ABB RobotStudio station: RS2_Picker.rsstn

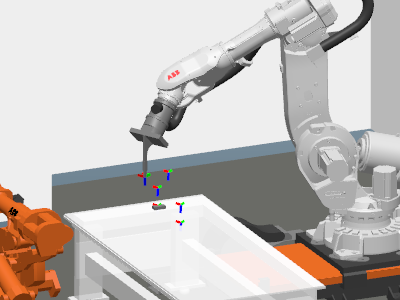
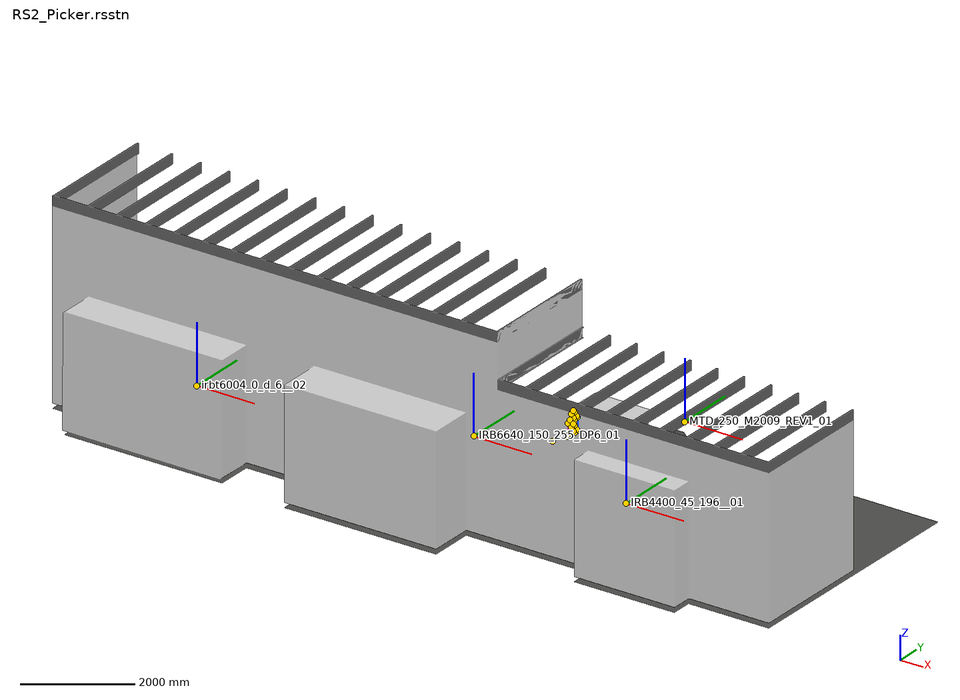
[picture v1: parts stored in the station drawn from their meshes, with robot base, taught points and paths (robot models come from the ABB library and are not in the file)]
Station RS2_Picker (saved by RobotStudio 22.2.9947.0)
Controller dFAB4400, task T_ROB1: task frame (RAPID world) sits at (8239.64, -6.06, -391.24) mm, rotated rx 0 ry 0 rz 180 deg in the station
Controller 66-101898AOFFLINE
  mechanical unit TRACK_1: irbt6004_0_d_6__02, 1 joints, base frame (0, 0, 0) mm
  mechanical unit ROB_1: IRB6640_150_255_DP6_01, 6 joints, base frame (0, 0, 0) mm
Controller dFAB4400
  mechanical unit STN1: MTD_250_M2009_REV1_01, 1 joints, base frame (1410.71, 486.5, 778.9) mm, rotated rx 0 ry 0 rz 90 deg
  mechanical unit ROB_1: IRB4400_45_196__01, 6 joints, base frame (0, 0, 0) mm
Layout (positions relative to the parent item):
  - irbt6004_0_d_6__02 [mechanism, from Libraries\irbt6004_0_d_6__02.rslib] at (-550.5, -475, -384.5) mm; joint values [5] (rad or m)
  - IRB6640_150_255_DP6_01 [mechanism, from Libraries\IRB6640_150_255_DP6_G_01.rslib] at (5000, 0, 0) mm; joint values [-0.2102, 0.1488, 0.3671, 0.9174, 0.6091, -0.3077] (rad or m)
  - rotary_stand [part], size 301.9 x 311.7 x 727.3 mm
  - MTD_250_M2009_REV1_01 [mechanism, from Libraries\MTD_250_M2009_REV1_01.rslib] at (8228.8, 1787.55, 468) mm, rotated rx 0 ry 0 rz 90 deg; joint values [0] (rad or m)
  - IRB4400_45_196__01 [mechanism, from Robots\IRB4400_45_196__01.rslib] at (8239.64, -6.06, -391.24) mm, rotated rx 0 ry 0 rz 180 deg; joint values [1.5707, -1.1345, 0, 0, 0, 0] (rad or m)
  - aarl_floor [part] at (0, 0, -101) mm, size 15367 x 6261.1 x 0 mm
  - 4400 ATI [part] at (8239.59, -419.45, 814.89) mm, rotated rx 0 ry 90 rz -90.01 deg, size 369.5 x 443 x 336 mm
  - AARL_Walls_west [part], size 15367 x 3481.8 x 3810 mm
  - AARL_Walls_east [part], size 15367 x 2779.3 x 3810 mm
  - AARL_Ceiling_west [part], size 15214.6 x 2567.4 x 1117.6 mm
  - VaccumTable_AtEndOfTrack [part], size 1240.6 x 2443.9 x 841 mm
  - ExpanderStation [part], size 715.1 x 918.2 x 79.1 mm
  - Component_SteelTable_2015_10_31 [part] at (1803.71, -1743.4, 287.57) mm, rotated rx 0.58 ry -0.13 rz 179.69 deg, size 2772.7 x 1553.5 x 641.4 mm
  - 20151025_RobotBar_2 [part] at (10163.42, -1202.89, 872.63) mm, rotated rx -90.3 ry 0.37 rz -90.64 deg, size 3760 x 1271.6 x 704 mm
  - 20151107_6640Table_andAlcove [part] at (1803.71, -1743.4, 287.57) mm, rotated rx 0.58 ry -0.13 rz 179.69 deg, size 3362 x 1558.7 x 2265 mm
  - Cameras In Alcove [part], size 3672.3 x 1646.1 x 329.3 mm
  - 6640 ATI [part] at (6755.25, -212.35, 1206.62) mm, rotated rx 139.11 ry 20.7 rz 140.14 deg, size 185.4 x 185.4 x 86.9 mm
  - suctionGripperTool [mechanism] at (6755.25, -212.35, 1206.62) mm, rotated rx 139.11 ry 20.7 rz 140.14 deg
      TCP suctionGripperTool at (-65.22, 118.54, 382.24) mm, rotated rx -42.17 ry -15.36 rz 13.49 deg
      links: Dummy
  - Part_1 [part] at (6893.07, 6354.78, 0) mm, rotated rx 0 ry 0 rz -90.01 deg, size 50 x 100 x 25 mm
  - ITARF23_Pincher [mechanism] at (6755.25, -212.35, 1206.62) mm, rotated rx -139.11 ry -20.7 rz -39.86 deg
      TCP ITARF23_Pincher at (-65.22, 118.54, 382.24) mm, rotated rx -42.17 ry -15.36 rz 13.49 deg
      links: pincherTool
Attachment: IRB6640_150_255_DP6_01 is attached to irbt6004_0_d_6__02 / Link1
Attachment: 4400 ATI is attached to IRB4400_45_196__01 / Link6
Attachment: 6640 ATI is attached to IRB6640_150_255_DP6_01 / Link6
Attachment: suctionGripperTool is attached to IRB6640_150_255_DP6_01 / Link6
Attachment: ITARF23_Pincher is attached to IRB6640_150_255_DP6_01 / Link6
Collision set CollisionSet_1: 4400 ATI against Link4, Link2, near miss 0 m
Collision set CollisionSet_2: 20151025_RobotBar_2 against IRB4400_45_196__01, near miss 0.005 m
Collision set CollisionSet_3: 20151107_6640Table_andAlcove, Component_SteelTable_2015_10_31, ExpanderStation against IRB6640_150_255_DP6_01, near miss 0.005 m
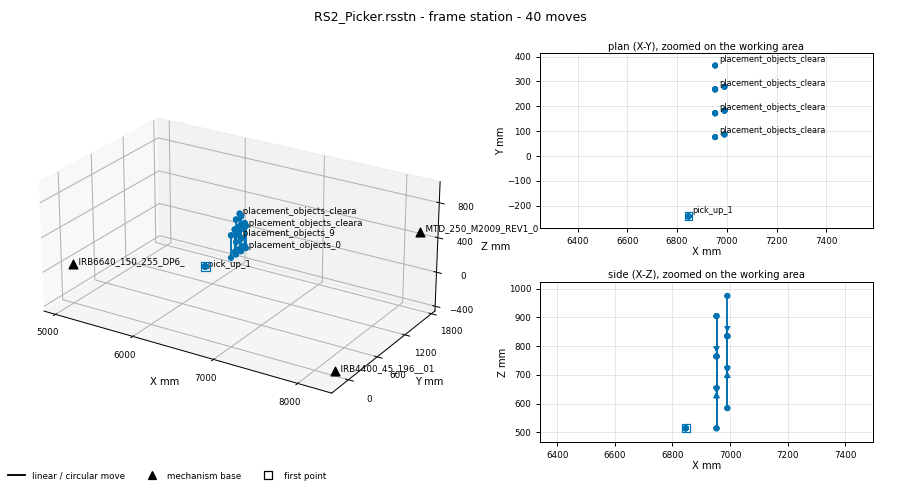
[picture p0: tool path of RS2_Picker.rsstn in frame station, 40 of 72 moves have a stored position in this frame; points joined in program order, loops and branches not executed]
Targets, tools, work objects and paths stored in the station, written as RAPID:
! task T_ROB1
MODULE Inc_Form_Test_090816
  VAR speeddata mySpeed:=[250,250,5000,1000];
  VAR zonedata myZone:=[FALSE,5,5,10,5,10,3];
ENDMODULE

! task T_ROB1
MODULE RobotProgramModule
  CONST robtarget t_pick:=[[6693.807660738,-323.119608005,453.981396454],[0.055399765,0.879680571,-0.471265936,0.031644522],[-1,0,-3,0],[4333.256617002,9E+09,9E+09,9E+09,9E+09,9E+09]];
  CONST robtarget t_pick_safe:=[[6693.807675418,-323.1195903,606.653821091],[0.055399731,0.879680578,-0.471265927,0.031644523],[-1,0,-2,0],[4333.256617002,9E+09,9E+09,9E+09,9E+09,9E+09]];
  CONST robtarget t_place_safe:=[[6693.807761035,133.958968301,606.65379018],[0.05539974,0.879680599,-0.471265883,0.031644591],[0,-1,-2,0],[4333.256617002,9E+09,9E+09,9E+09,9E+09,9E+09]];
  CONST robtarget t_place:=[[6693.80755977,133.959044617,452.547726462],[0.055399551,0.879680524,-0.471266043,0.031644636],[0,-1,-2,0],[4333.256617002,9E+09,9E+09,9E+09,9E+09,9E+09]];
  CONST robtarget t_home:=[[6693.807553504,-112.078129424,808.817014857],[0.055399679,0.879680616,-0.471265852,0.031644705],[-1,0,-2,0],[4333.256617002,9E+09,9E+09,9E+09,9E+09,9E+09]];
ENDMODULE

! task T_ROB1
MODULE CalibData
  PERS tooldata ITARF23_Pincher:=[TRUE,[[-65.2151,118.542,382.236],[0.180955748,0.120020452,-0.358114493,-0.908077155]],[1,[0,0,1],[1,0,0,0],0,0,0]];
ENDMODULE

! task T_ROB1
MODULE MainModule
  PERS tooldata two_finger_gripper_itar2:=[TRUE,[[94.35,-163.419,405.705],[-0.239118,0.099041,-0.369628,0.892406]],[0.001,[0,0,0.001],[1,0,0,0],0,0,0]];
  VAR jointtarget pos_home:=[[1,2,3,4,5,6],[4200,9E+09,9E+09,9E+09,9E+09,9E+09]];
  VAR robtarget pick_up_1:=[[6845.94,-242.64,514.59],[0,0.707107,-0.707107,0],[0,0,0,0],[5000,9E+09,9E+09,9E+09,9E+09,9E+09]];
  VAR robtarget placement_objects_clearance_0:=[[6952.98,364.03,764.59],[0,0.707107,-0.707107,0],[0,0,0,0],[5000,9E+09,9E+09,9E+09,9E+09,9E+09]];
  VAR robtarget placement_objects_0:=[[6952.98,364.03,514.59],[0,0.707107,-0.707107,0],[0,0,0,0],[5000,9E+09,9E+09,9E+09,9E+09,9E+09]];
  VAR robtarget placement_objects_clearance_1:=[[6952.98,268.03,764.59],[0,0.707107,-0.707107,0],[0,0,0,0],[5000,9E+09,9E+09,9E+09,9E+09,9E+09]];
  VAR robtarget placement_objects_1:=[[6952.98,268.03,514.59],[0,0.707107,-0.707107,0],[0,0,0,0],[5000,9E+09,9E+09,9E+09,9E+09,9E+09]];
  VAR robtarget placement_objects_clearance_2:=[[6952.98,172.03,764.59],[0,0.707107,-0.707107,0],[0,0,0,0],[5000,9E+09,9E+09,9E+09,9E+09,9E+09]];
  VAR robtarget placement_objects_2:=[[6952.98,172.03,514.59],[0,0.707107,-0.707107,0],[0,0,0,0],[5000,9E+09,9E+09,9E+09,9E+09,9E+09]];
  VAR robtarget placement_objects_clearance_3:=[[6952.98,76.03,764.59],[0,0.707107,-0.707107,0],[0,0,0,0],[5000,9E+09,9E+09,9E+09,9E+09,9E+09]];
  VAR robtarget placement_objects_3:=[[6952.98,76.03,514.59],[0,0.707107,-0.707107,0],[0,0,0,0],[5000,9E+09,9E+09,9E+09,9E+09,9E+09]];
  VAR robtarget placement_objects_clearance_4:=[[6990.48,278.53,834.59],[0,1,0,0],[0,0,0,0],[5000,9E+09,9E+09,9E+09,9E+09,9E+09]];
  VAR robtarget placement_objects_4:=[[6990.48,278.53,584.59],[0,1,0,0],[0,0,0,0],[5000,9E+09,9E+09,9E+09,9E+09,9E+09]];
  VAR robtarget placement_objects_clearance_5:=[[6990.48,182.53,834.59],[0,1,0,0],[0,0,0,0],[5000,9E+09,9E+09,9E+09,9E+09,9E+09]];
  VAR robtarget placement_objects_5:=[[6990.48,182.53,584.59],[0,1,0,0],[0,0,0,0],[5000,9E+09,9E+09,9E+09,9E+09,9E+09]];
  VAR robtarget placement_objects_clearance_6:=[[6990.48,86.53,834.59],[0,1,0,0],[0,0,0,0],[5000,9E+09,9E+09,9E+09,9E+09,9E+09]];
  VAR robtarget placement_objects_6:=[[6990.48,86.53,584.59],[0,1,0,0],[0,0,0,0],[5000,9E+09,9E+09,9E+09,9E+09,9E+09]];
  VAR robtarget placement_objects_clearance_7:=[[6952.98,268.03,904.59],[0,0.707107,-0.707107,0],[0,0,0,0],[5000,9E+09,9E+09,9E+09,9E+09,9E+09]];
  VAR robtarget placement_objects_7:=[[6952.98,268.03,654.59],[0,0.707107,-0.707107,0],[0,0,0,0],[5000,9E+09,9E+09,9E+09,9E+09,9E+09]];
  VAR robtarget placement_objects_clearance_8:=[[6952.98,172.03,904.59],[0,0.707107,-0.707107,0],[0,0,0,0],[5000,9E+09,9E+09,9E+09,9E+09,9E+09]];
  VAR robtarget placement_objects_8:=[[6952.98,172.03,654.59],[0,0.707107,-0.707107,0],[0,0,0,0],[5000,9E+09,9E+09,9E+09,9E+09,9E+09]];
  VAR robtarget placement_objects_clearance_9:=[[6990.48,182.53,974.59],[0,1,0,0],[0,0,0,0],[5000,9E+09,9E+09,9E+09,9E+09,9E+09]];
  VAR robtarget placement_objects_9:=[[6990.48,182.53,724.59],[0,1,0,0],[0,0,0,0],[5000,9E+09,9E+09,9E+09,9E+09,9E+09]];
  PROC new_pincher()
    ConfJ \On;
    MoveAbsJ pos_home,v200,z50,two_finger_gripper_itar2\WObj:=wobj0;
    ConfJ \Off;
    ConfJ \On;
    MoveAbsJ pos_home,v200,z50,two_finger_gripper_itar2\WObj:=wobj0;
    ConfJ \Off;
    WaitTime 1;
    SetDO do_tool_gripper_close,0;
    SetDO do_tool_gripper_open,1;
    WaitTime 2;
    MoveJ il_21,v300,z15,two_finger_gripper_itar2\WObj:=wobj0;
    MoveL pick_up_1,v300,z0,two_finger_gripper_itar2\WObj:=wobj0;
    WaitTime 1;
    SetDO do_tool_gripper_close,1;
    SetDO do_tool_gripper_open,0;
    WaitTime 2;
    MoveJ il_22,v300,z15,two_finger_gripper_itar2\WObj:=wobj0;
    MoveL placement_objects_clearance_0,v300,z0,two_finger_gripper_itar2\WObj:=wobj0;
    MoveL placement_objects_0,v300,z0,two_finger_gripper_itar2\WObj:=wobj0;
    WaitTime 1;
    SetDO do_tool_gripper_close,0;
    SetDO do_tool_gripper_open,1;
    WaitTime 2;
    MoveL placement_objects_clearance_0,v150,z0,two_finger_gripper_itar2\WObj:=wobj0;
    ConfJ \On;
    MoveAbsJ pos_home,v200,z50,two_finger_gripper_itar2\WObj:=wobj0;
    ConfJ \Off;
    WaitTime 1;
    SetDO do_tool_gripper_close,0;
    SetDO do_tool_gripper_open,1;
    WaitTime 2;
    MoveJ il_23,v300,z15,two_finger_gripper_itar2\WObj:=wobj0;
    MoveL pick_up_1,v300,z0,two_finger_gripper_itar2\WObj:=wobj0;
    WaitTime 1;
    SetDO do_tool_gripper_close,1;
    SetDO do_tool_gripper_open,0;
    WaitTime 2;
    MoveJ il_24,v300,z15,two_finger_gripper_itar2\WObj:=wobj0;
    MoveL placement_objects_clearance_1,v300,z0,two_finger_gripper_itar2\WObj:=wobj0;
    MoveL placement_objects_1,v300,z0,two_finger_gripper_itar2\WObj:=wobj0;
    WaitTime 1;
    SetDO do_tool_gripper_close,0;
    SetDO do_tool_gripper_open,1;
    WaitTime 2;
    MoveL placement_objects_clearance_1,v150,z0,two_finger_gripper_itar2\WObj:=wobj0;
    ConfJ \On;
    MoveAbsJ pos_home,v200,z50,two_finger_gripper_itar2\WObj:=wobj0;
    ConfJ \Off;
    WaitTime 1;
    SetDO do_tool_gripper_close,0;
    SetDO do_tool_gripper_open,1;
    WaitTime 2;
    MoveJ il_25,v300,z15,two_finger_gripper_itar2\WObj:=wobj0;
    MoveL pick_up_1,v300,z0,two_finger_gripper_itar2\WObj:=wobj0;
    WaitTime 1;
    SetDO do_tool_gripper_close,1;
    SetDO do_tool_gripper_open,0;
    WaitTime 2;
    MoveJ il_26,v300,z15,two_finger_gripper_itar2\WObj:=wobj0;
    MoveL placement_objects_clearance_2,v300,z0,two_finger_gripper_itar2\WObj:=wobj0;
    MoveL placement_objects_2,v300,z0,two_finger_gripper_itar2\WObj:=wobj0;
    WaitTime 1;
    SetDO do_tool_gripper_close,0;
    SetDO do_tool_gripper_open,1;
    WaitTime 2;
    MoveL placement_objects_clearance_2,v150,z0,two_finger_gripper_itar2\WObj:=wobj0;
    ConfJ \On;
    MoveAbsJ pos_home,v200,z50,two_finger_gripper_itar2\WObj:=wobj0;
    ConfJ \Off;
    WaitTime 1;
    SetDO do_tool_gripper_close,0;
    SetDO do_tool_gripper_open,1;
    WaitTime 2;
    MoveJ il_27,v300,z15,two_finger_gripper_itar2\WObj:=wobj0;
    MoveL pick_up_1,v300,z0,two_finger_gripper_itar2\WObj:=wobj0;
    WaitTime 1;
    SetDO do_tool_gripper_close,1;
    SetDO do_tool_gripper_open,0;
    WaitTime 2;
    MoveJ il_28,v300,z15,two_finger_gripper_itar2\WObj:=wobj0;
    MoveL placement_objects_clearance_3,v300,z0,two_finger_gripper_itar2\WObj:=wobj0;
    MoveL placement_objects_3,v300,z0,two_finger_gripper_itar2\WObj:=wobj0;
    WaitTime 1;
    SetDO do_tool_gripper_close,0;
    SetDO do_tool_gripper_open,1;
    WaitTime 2;
    MoveL placement_objects_clearance_3,v150,z0,two_finger_gripper_itar2\WObj:=wobj0;
    ConfJ \On;
    MoveAbsJ pos_home,v200,z50,two_finger_gripper_itar2\WObj:=wobj0;
    ConfJ \Off;
    WaitTime 1;
    SetDO do_tool_gripper_close,0;
    SetDO do_tool_gripper_open,1;
    WaitTime 2;
    MoveJ il_29,v300,z15,two_finger_gripper_itar2\WObj:=wobj0;
    MoveL pick_up_1,v300,z0,two_finger_gripper_itar2\WObj:=wobj0;
    WaitTime 1;
    SetDO do_tool_gripper_close,1;
    SetDO do_tool_gripper_open,0;
    WaitTime 2;
    MoveJ il_30,v300,z15,two_finger_gripper_itar2\WObj:=wobj0;
    MoveL placement_objects_clearance_4,v300,z0,two_finger_gripper_itar2\WObj:=wobj0;
    MoveL placement_objects_4,v300,z0,two_finger_gripper_itar2\WObj:=wobj0;
    WaitTime 1;
    SetDO do_tool_gripper_close,0;
    SetDO do_tool_gripper_open,1;
    WaitTime 2;
    MoveL placement_objects_clearance_4,v150,z0,two_finger_gripper_itar2\WObj:=wobj0;
    ConfJ \On;
    MoveAbsJ pos_home,v200,z50,two_finger_gripper_itar2\WObj:=wobj0;
    ConfJ \Off;
    WaitTime 1;
    SetDO do_tool_gripper_close,0;
    SetDO do_tool_gripper_open,1;
    WaitTime 2;
    MoveJ il_31,v300,z15,two_finger_gripper_itar2\WObj:=wobj0;
    MoveL pick_up_1,v300,z0,two_finger_gripper_itar2\WObj:=wobj0;
    WaitTime 1;
    SetDO do_tool_gripper_close,1;
    SetDO do_tool_gripper_open,0;
    WaitTime 2;
    MoveJ il_32,v300,z15,two_finger_gripper_itar2\WObj:=wobj0;
    MoveL placement_objects_clearance_5,v300,z0,two_finger_gripper_itar2\WObj:=wobj0;
    MoveL placement_objects_5,v300,z0,two_finger_gripper_itar2\WObj:=wobj0;
    WaitTime 1;
    SetDO do_tool_gripper_close,0;
    SetDO do_tool_gripper_open,1;
    WaitTime 2;
    MoveL placement_objects_clearance_5,v150,z0,two_finger_gripper_itar2\WObj:=wobj0;
    ConfJ \On;
    MoveAbsJ pos_home,v200,z50,two_finger_gripper_itar2\WObj:=wobj0;
    ConfJ \Off;
    WaitTime 1;
    SetDO do_tool_gripper_close,0;
    SetDO do_tool_gripper_open,1;
    WaitTime 2;
    MoveJ il_33,v300,z15,two_finger_gripper_itar2\WObj:=wobj0;
    MoveL pick_up_1,v300,z0,two_finger_gripper_itar2\WObj:=wobj0;
    WaitTime 1;
    SetDO do_tool_gripper_close,1;
    SetDO do_tool_gripper_open,0;
    WaitTime 2;
    MoveJ il_34,v300,z15,two_finger_gripper_itar2\WObj:=wobj0;
    MoveL placement_objects_clearance_6,v300,z0,two_finger_gripper_itar2\WObj:=wobj0;
    MoveL placement_objects_6,v300,z0,two_finger_gripper_itar2\WObj:=wobj0;
    WaitTime 1;
    SetDO do_tool_gripper_close,0;
    SetDO do_tool_gripper_open,1;
    WaitTime 2;
    MoveL placement_objects_clearance_6,v150,z0,two_finger_gripper_itar2\WObj:=wobj0;
    ConfJ \On;
    MoveAbsJ pos_home,v200,z50,two_finger_gripper_itar2\WObj:=wobj0;
    ConfJ \Off;
    WaitTime 1;
    SetDO do_tool_gripper_close,0;
    SetDO do_tool_gripper_open,1;
    WaitTime 2;
    MoveJ il_35,v300,z15,two_finger_gripper_itar2\WObj:=wobj0;
    MoveL pick_up_1,v300,z0,two_finger_gripper_itar2\WObj:=wobj0;
    WaitTime 1;
    SetDO do_tool_gripper_close,1;
    SetDO do_tool_gripper_open,0;
    WaitTime 2;
    MoveJ il_36,v300,z15,two_finger_gripper_itar2\WObj:=wobj0;
    MoveL placement_objects_clearance_7,v300,z0,two_finger_gripper_itar2\WObj:=wobj0;
    MoveL placement_objects_7,v300,z0,two_finger_gripper_itar2\WObj:=wobj0;
    WaitTime 1;
    SetDO do_tool_gripper_close,0;
    SetDO do_tool_gripper_open,1;
    WaitTime 2;
    MoveL placement_objects_clearance_7,v150,z0,two_finger_gripper_itar2\WObj:=wobj0;
    ConfJ \On;
    MoveAbsJ pos_home,v200,z50,two_finger_gripper_itar2\WObj:=wobj0;
    ConfJ \Off;
    WaitTime 1;
    SetDO do_tool_gripper_close,0;
    SetDO do_tool_gripper_open,1;
    WaitTime 2;
    MoveJ il_37,v300,z15,two_finger_gripper_itar2\WObj:=wobj0;
    MoveL pick_up_1,v300,z0,two_finger_gripper_itar2\WObj:=wobj0;
    WaitTime 1;
    SetDO do_tool_gripper_close,1;
    SetDO do_tool_gripper_open,0;
    WaitTime 2;
    MoveJ il_38,v300,z15,two_finger_gripper_itar2\WObj:=wobj0;
    MoveL placement_objects_clearance_8,v300,z0,two_finger_gripper_itar2\WObj:=wobj0;
    MoveL placement_objects_8,v300,z0,two_finger_gripper_itar2\WObj:=wobj0;
    WaitTime 1;
    SetDO do_tool_gripper_close,0;
    SetDO do_tool_gripper_open,1;
    WaitTime 2;
    MoveL placement_objects_clearance_8,v150,z0,two_finger_gripper_itar2\WObj:=wobj0;
    ConfJ \On;
    MoveAbsJ pos_home,v200,z50,two_finger_gripper_itar2\WObj:=wobj0;
    ConfJ \Off;
    WaitTime 1;
    SetDO do_tool_gripper_close,0;
    SetDO do_tool_gripper_open,1;
    WaitTime 2;
    MoveJ il_39,v300,z15,two_finger_gripper_itar2\WObj:=wobj0;
    MoveL pick_up_1,v300,z0,two_finger_gripper_itar2\WObj:=wobj0;
    WaitTime 1;
    SetDO do_tool_gripper_close,1;
    SetDO do_tool_gripper_open,0;
    WaitTime 2;
    MoveJ il_40,v300,z15,two_finger_gripper_itar2\WObj:=wobj0;
    MoveL placement_objects_clearance_9,v300,z0,two_finger_gripper_itar2\WObj:=wobj0;
    MoveL placement_objects_9,v300,z0,two_finger_gripper_itar2\WObj:=wobj0;
    WaitTime 1;
    SetDO do_tool_gripper_close,0;
    SetDO do_tool_gripper_open,1;
    WaitTime 2;
    MoveL placement_objects_clearance_9,v150,z0,two_finger_gripper_itar2\WObj:=wobj0;
    ConfJ \On;
    MoveAbsJ pos_home,v200,z50,two_finger_gripper_itar2\WObj:=wobj0;
    ConfJ \Off;
  ENDPROC
ENDMODULE

